// TIA Portal V19 export
FUNCTION "PREMIXING TRANSFER CYCLE" : Void   // FC25, LAD
{ S7_Optimized_Access := 'TRUE' }
// stored: SetENOAutomatically false
   VAR_TEMP   // added for the SCL form of the ladder/FBD networks
      _w1 : Bool;
   END_VAR
BEGIN

REGION Network 1: TRANSFER SELECT
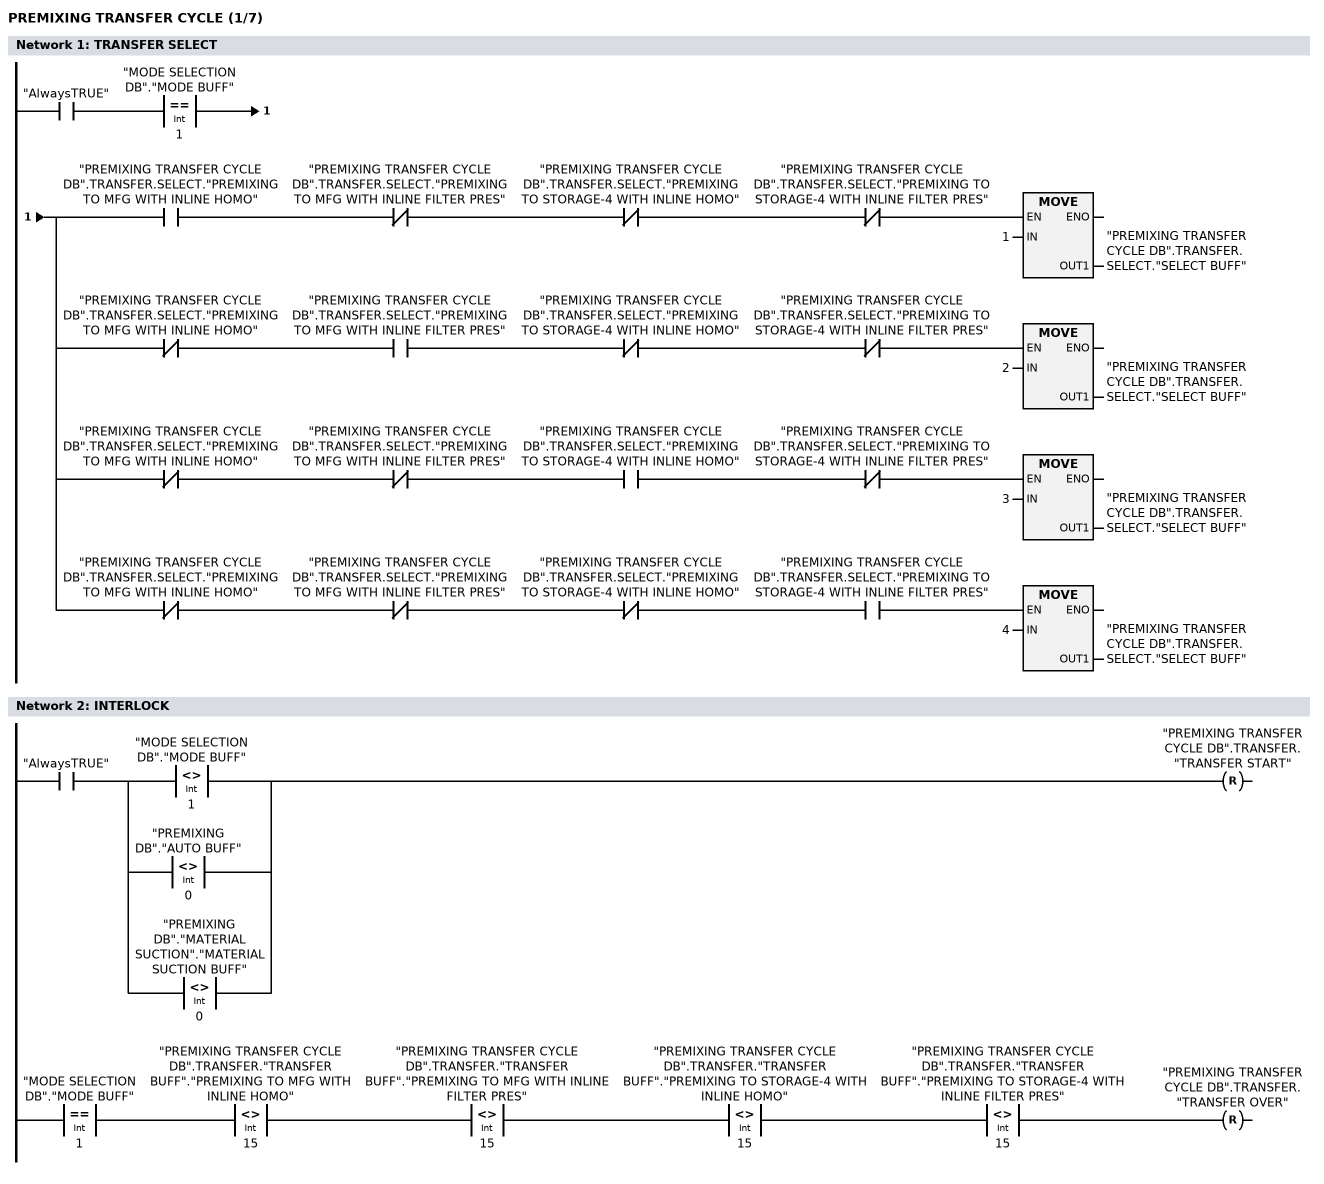
   RUNG wire#powerrail
      Contact( "AlwaysTRUE" )
      { S7_Templates := "SrcType := Int" } EQ_Contact(in1 := "MODE SELECTION DB"."MODE BUFF", in2 := 1)
      wire#w1
      Contact( "PREMIXING TRANSFER CYCLE DB".TRANSFER.SELECT."PREMIXING TO MFG WITH INLINE HOMO" )
      I_Contact( "PREMIXING TRANSFER CYCLE DB".TRANSFER.SELECT."PREMIXING TO MFG WITH INLINE FILTER PRES" )
      I_Contact( "PREMIXING TRANSFER CYCLE DB".TRANSFER.SELECT."PREMIXING TO STORAGE-4 WITH INLINE HOMO" )
      I_Contact( "PREMIXING TRANSFER CYCLE DB".TRANSFER.SELECT."PREMIXING TO STORAGE-4 WITH INLINE FILTER PRES" )
      Move(in := 1, out1 => "PREMIXING TRANSFER CYCLE DB".TRANSFER.SELECT."SELECT BUFF")
   END_RUNG
   RUNG wire#w1
      I_Contact( "PREMIXING TRANSFER CYCLE DB".TRANSFER.SELECT."PREMIXING TO MFG WITH INLINE HOMO" )
      Contact( "PREMIXING TRANSFER CYCLE DB".TRANSFER.SELECT."PREMIXING TO MFG WITH INLINE FILTER PRES" )
      I_Contact( "PREMIXING TRANSFER CYCLE DB".TRANSFER.SELECT."PREMIXING TO STORAGE-4 WITH INLINE HOMO" )
      I_Contact( "PREMIXING TRANSFER CYCLE DB".TRANSFER.SELECT."PREMIXING TO STORAGE-4 WITH INLINE FILTER PRES" )
      Move(in := 2, out1 => "PREMIXING TRANSFER CYCLE DB".TRANSFER.SELECT."SELECT BUFF")
   END_RUNG
   RUNG wire#w1
      I_Contact( "PREMIXING TRANSFER CYCLE DB".TRANSFER.SELECT."PREMIXING TO MFG WITH INLINE HOMO" )
      I_Contact( "PREMIXING TRANSFER CYCLE DB".TRANSFER.SELECT."PREMIXING TO MFG WITH INLINE FILTER PRES" )
      Contact( "PREMIXING TRANSFER CYCLE DB".TRANSFER.SELECT."PREMIXING TO STORAGE-4 WITH INLINE HOMO" )
      I_Contact( "PREMIXING TRANSFER CYCLE DB".TRANSFER.SELECT."PREMIXING TO STORAGE-4 WITH INLINE FILTER PRES" )
      Move(in := 3, out1 => "PREMIXING TRANSFER CYCLE DB".TRANSFER.SELECT."SELECT BUFF")
   END_RUNG
   RUNG wire#w1
      I_Contact( "PREMIXING TRANSFER CYCLE DB".TRANSFER.SELECT."PREMIXING TO MFG WITH INLINE HOMO" )
      I_Contact( "PREMIXING TRANSFER CYCLE DB".TRANSFER.SELECT."PREMIXING TO MFG WITH INLINE FILTER PRES" )
      I_Contact( "PREMIXING TRANSFER CYCLE DB".TRANSFER.SELECT."PREMIXING TO STORAGE-4 WITH INLINE HOMO" )
      Contact( "PREMIXING TRANSFER CYCLE DB".TRANSFER.SELECT."PREMIXING TO STORAGE-4 WITH INLINE FILTER PRES" )
      Move(in := 4, out1 => "PREMIXING TRANSFER CYCLE DB".TRANSFER.SELECT."SELECT BUFF")
   END_RUNG
   // the same network as SCL:
   #_w1 := "AlwaysTRUE" AND ("MODE SELECTION DB"."MODE BUFF" = 1);
   IF #_w1 AND "PREMIXING TRANSFER CYCLE DB".TRANSFER.SELECT."PREMIXING TO MFG WITH INLINE HOMO" AND NOT "PREMIXING TRANSFER CYCLE DB".TRANSFER.SELECT."PREMIXING TO MFG WITH INLINE FILTER PRES" AND NOT "PREMIXING TRANSFER CYCLE DB".TRANSFER.SELECT."PREMIXING TO STORAGE-4 WITH INLINE HOMO" AND NOT "PREMIXING TRANSFER CYCLE DB".TRANSFER.SELECT."PREMIXING TO STORAGE-4 WITH INLINE FILTER PRES" THEN
       "PREMIXING TRANSFER CYCLE DB".TRANSFER.SELECT."SELECT BUFF" := 1;
   END_IF;
   IF #_w1 AND NOT "PREMIXING TRANSFER CYCLE DB".TRANSFER.SELECT."PREMIXING TO MFG WITH INLINE HOMO" AND "PREMIXING TRANSFER CYCLE DB".TRANSFER.SELECT."PREMIXING TO MFG WITH INLINE FILTER PRES" AND NOT "PREMIXING TRANSFER CYCLE DB".TRANSFER.SELECT."PREMIXING TO STORAGE-4 WITH INLINE HOMO" AND NOT "PREMIXING TRANSFER CYCLE DB".TRANSFER.SELECT."PREMIXING TO STORAGE-4 WITH INLINE FILTER PRES" THEN
       "PREMIXING TRANSFER CYCLE DB".TRANSFER.SELECT."SELECT BUFF" := 2;
   END_IF;
   IF #_w1 AND NOT "PREMIXING TRANSFER CYCLE DB".TRANSFER.SELECT."PREMIXING TO MFG WITH INLINE HOMO" AND NOT "PREMIXING TRANSFER CYCLE DB".TRANSFER.SELECT."PREMIXING TO MFG WITH INLINE FILTER PRES" AND "PREMIXING TRANSFER CYCLE DB".TRANSFER.SELECT."PREMIXING TO STORAGE-4 WITH INLINE HOMO" AND NOT "PREMIXING TRANSFER CYCLE DB".TRANSFER.SELECT."PREMIXING TO STORAGE-4 WITH INLINE FILTER PRES" THEN
       "PREMIXING TRANSFER CYCLE DB".TRANSFER.SELECT."SELECT BUFF" := 3;
   END_IF;
   IF #_w1 AND NOT "PREMIXING TRANSFER CYCLE DB".TRANSFER.SELECT."PREMIXING TO MFG WITH INLINE HOMO" AND NOT "PREMIXING TRANSFER CYCLE DB".TRANSFER.SELECT."PREMIXING TO MFG WITH INLINE FILTER PRES" AND NOT "PREMIXING TRANSFER CYCLE DB".TRANSFER.SELECT."PREMIXING TO STORAGE-4 WITH INLINE HOMO" AND "PREMIXING TRANSFER CYCLE DB".TRANSFER.SELECT."PREMIXING TO STORAGE-4 WITH INLINE FILTER PRES" THEN
       "PREMIXING TRANSFER CYCLE DB".TRANSFER.SELECT."SELECT BUFF" := 4;
   END_IF;
END_REGION

REGION Network 2: INTERLOCK
   RUNG wire#powerrail
      Contact( "AlwaysTRUE" )
      wire#w1
      { S7_Templates := "SrcType := Int" } NE_Contact(in1 := "MODE SELECTION DB"."MODE BUFF", in2 := 1)
      wire#w2
      R_Coil( "PREMIXING TRANSFER CYCLE DB".TRANSFER."TRANSFER START" )
   END_RUNG
   RUNG wire#w1
      { S7_Templates := "SrcType := Int" } NE_Contact(in1 := "PREMIXING DB"."AUTO BUFF", in2 := 0)
   END_RUNG wire#w2
   RUNG wire#w1
      { S7_Templates := "SrcType := Int" } NE_Contact(in1 := "PREMIXING DB"."MATERIAL SUCTION"."MATERIAL SUCTION BUFF", in2 := 0)
   END_RUNG wire#w2
   RUNG wire#powerrail
      { S7_Templates := "SrcType := Int" } EQ_Contact(in1 := "MODE SELECTION DB"."MODE BUFF", in2 := 1)
      { S7_Templates := "SrcType := Int" } NE_Contact(in1 := "PREMIXING TRANSFER CYCLE DB".TRANSFER."TRANSFER BUFF"."PREMIXING TO MFG WITH INLINE HOMO", in2 := 15)
      { S7_Templates := "SrcType := Int" } NE_Contact(in1 := "PREMIXING TRANSFER CYCLE DB".TRANSFER."TRANSFER BUFF"."PREMIXING TO MFG WITH INLINE FILTER PRES", in2 := 15)
      { S7_Templates := "SrcType := Int" } NE_Contact(in1 := "PREMIXING TRANSFER CYCLE DB".TRANSFER."TRANSFER BUFF"."PREMIXING TO STORAGE-4 WITH INLINE HOMO", in2 := 15)
      { S7_Templates := "SrcType := Int" } NE_Contact(in1 := "PREMIXING TRANSFER CYCLE DB".TRANSFER."TRANSFER BUFF"."PREMIXING TO STORAGE-4 WITH INLINE FILTER PRES", in2 := 15)
      R_Coil( "PREMIXING TRANSFER CYCLE DB".TRANSFER."TRANSFER OVER" )
   END_RUNG
   // the same network as SCL:
   IF "AlwaysTRUE" AND (("MODE SELECTION DB"."MODE BUFF" <> 1) OR ("PREMIXING DB"."AUTO BUFF" <> 0) OR ("PREMIXING DB"."MATERIAL SUCTION"."MATERIAL SUCTION BUFF" <> 0)) THEN
       "PREMIXING TRANSFER CYCLE DB".TRANSFER."TRANSFER START" := FALSE;
   END_IF;
   IF ("MODE SELECTION DB"."MODE BUFF" = 1) AND ("PREMIXING TRANSFER CYCLE DB".TRANSFER."TRANSFER BUFF"."PREMIXING TO MFG WITH INLINE HOMO" <> 15) AND ("PREMIXING TRANSFER CYCLE DB".TRANSFER."TRANSFER BUFF"."PREMIXING TO MFG WITH INLINE FILTER PRES" <> 15) AND ("PREMIXING TRANSFER CYCLE DB".TRANSFER."TRANSFER BUFF"."PREMIXING TO STORAGE-4 WITH INLINE HOMO" <> 15) AND ("PREMIXING TRANSFER CYCLE DB".TRANSFER."TRANSFER BUFF"."PREMIXING TO STORAGE-4 WITH INLINE FILTER PRES" <> 15) THEN
       "PREMIXING TRANSFER CYCLE DB".TRANSFER."TRANSFER OVER" := FALSE;
   END_IF;
END_REGION

REGION Network 3: TRANSFER START ///////////////////////////// PREMIXING TO MFG WITH INLINE HOMO
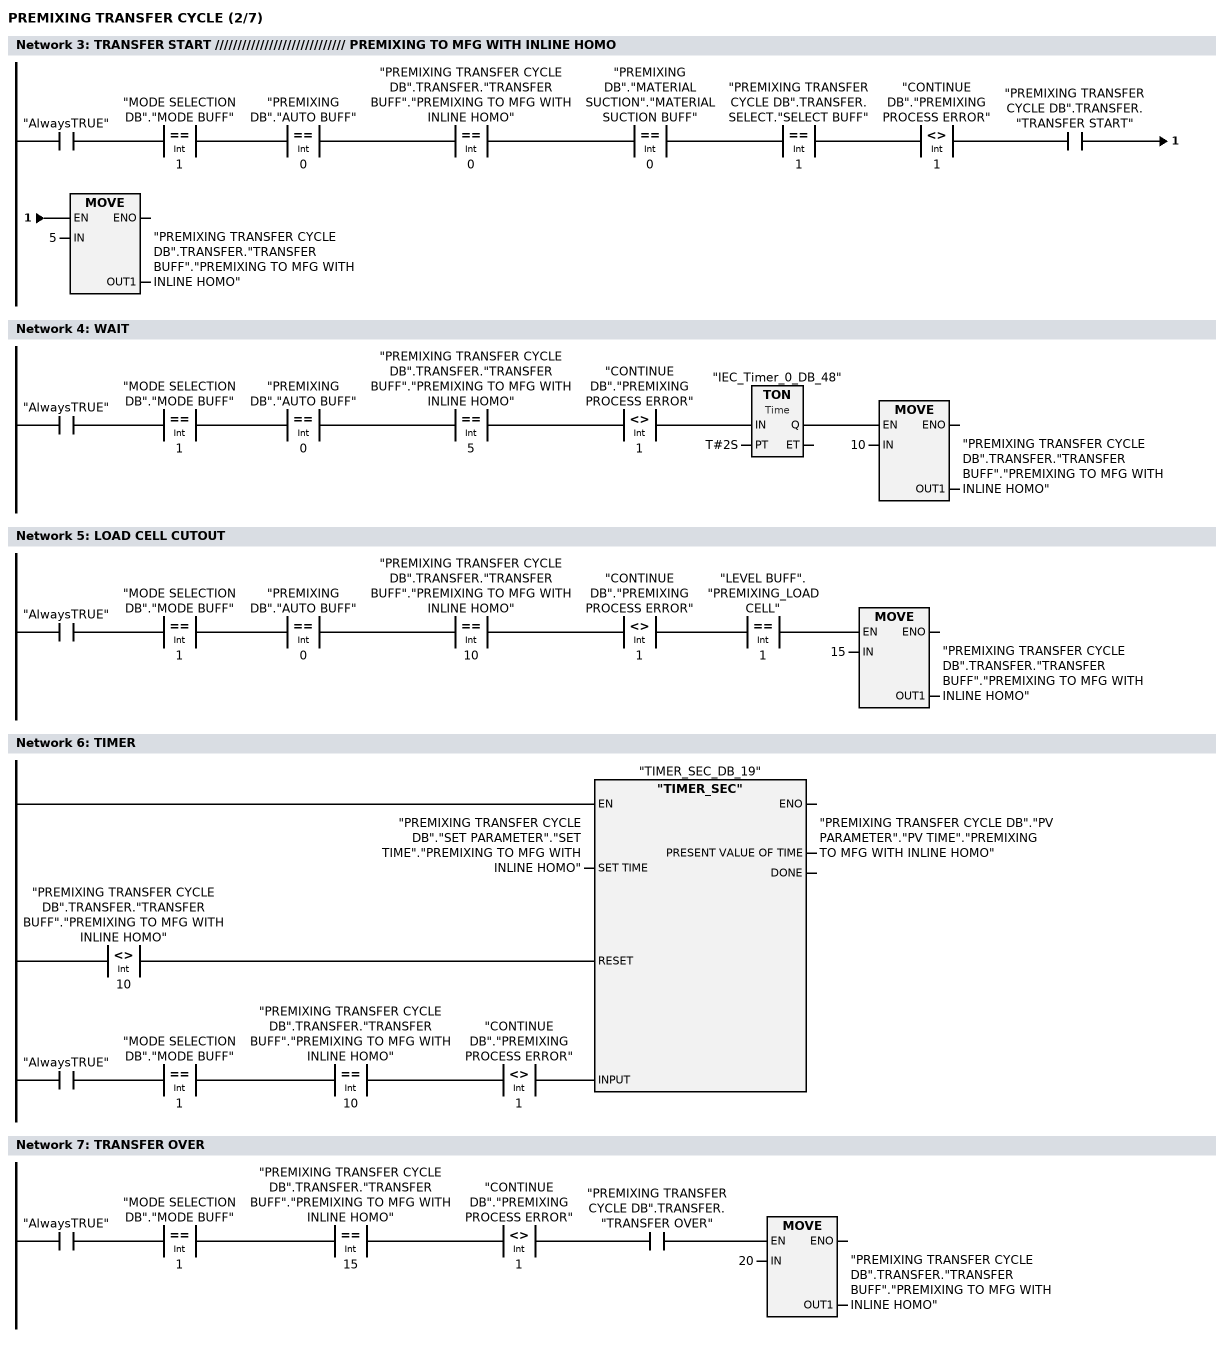
   RUNG wire#powerrail
      Contact( "AlwaysTRUE" )
      { S7_Templates := "SrcType := Int" } EQ_Contact(in1 := "MODE SELECTION DB"."MODE BUFF", in2 := 1)
      { S7_Templates := "SrcType := Int" } EQ_Contact(in1 := "PREMIXING DB"."AUTO BUFF", in2 := 0)
      { S7_Templates := "SrcType := Int" } EQ_Contact(in1 := "PREMIXING TRANSFER CYCLE DB".TRANSFER."TRANSFER BUFF"."PREMIXING TO MFG WITH INLINE HOMO", in2 := 0)
      { S7_Templates := "SrcType := Int" } EQ_Contact(in1 := "PREMIXING DB"."MATERIAL SUCTION"."MATERIAL SUCTION BUFF", in2 := 0)
      { S7_Templates := "SrcType := Int" } EQ_Contact(in1 := "PREMIXING TRANSFER CYCLE DB".TRANSFER.SELECT."SELECT BUFF", in2 := 1)
      { S7_Templates := "SrcType := Int" } NE_Contact(in1 := "CONTINUE DB"."PREMIXING PROCESS ERROR", in2 := 1)
      Contact( "PREMIXING TRANSFER CYCLE DB".TRANSFER."TRANSFER START" )
      Move(in := 5, out1 => "PREMIXING TRANSFER CYCLE DB".TRANSFER."TRANSFER BUFF"."PREMIXING TO MFG WITH INLINE HOMO")
   END_RUNG
   // the same network as SCL:
   IF "AlwaysTRUE" AND ("MODE SELECTION DB"."MODE BUFF" = 1) AND ("PREMIXING DB"."AUTO BUFF" = 0) AND ("PREMIXING TRANSFER CYCLE DB".TRANSFER."TRANSFER BUFF"."PREMIXING TO MFG WITH INLINE HOMO" = 0) AND ("PREMIXING DB"."MATERIAL SUCTION"."MATERIAL SUCTION BUFF" = 0) AND ("PREMIXING TRANSFER CYCLE DB".TRANSFER.SELECT."SELECT BUFF" = 1) AND ("CONTINUE DB"."PREMIXING PROCESS ERROR" <> 1) AND "PREMIXING TRANSFER CYCLE DB".TRANSFER."TRANSFER START" THEN
       "PREMIXING TRANSFER CYCLE DB".TRANSFER."TRANSFER BUFF"."PREMIXING TO MFG WITH INLINE HOMO" := 5;
   END_IF;
END_REGION

REGION Network 4: WAIT
   RUNG wire#powerrail
      Contact( "AlwaysTRUE" )
      { S7_Templates := "SrcType := Int" } EQ_Contact(in1 := "MODE SELECTION DB"."MODE BUFF", in2 := 1)
      { S7_Templates := "SrcType := Int" } EQ_Contact(in1 := "PREMIXING DB"."AUTO BUFF", in2 := 0)
      { S7_Templates := "SrcType := Int" } EQ_Contact(in1 := "PREMIXING TRANSFER CYCLE DB".TRANSFER."TRANSFER BUFF"."PREMIXING TO MFG WITH INLINE HOMO", in2 := 5)
      { S7_Templates := "SrcType := Int" } NE_Contact(in1 := "CONTINUE DB"."PREMIXING PROCESS ERROR", in2 := 1)
      { S7_Templates := "time_type := Time" } "IEC_Timer_0_DB_48".TON(pt := T#2S, et =>)
      Move(in := 10, out1 => "PREMIXING TRANSFER CYCLE DB".TRANSFER."TRANSFER BUFF"."PREMIXING TO MFG WITH INLINE HOMO")
   END_RUNG
   // the same network as SCL:
   "IEC_Timer_0_DB_48".TON(IN := "AlwaysTRUE" AND ("MODE SELECTION DB"."MODE BUFF" = 1) AND ("PREMIXING DB"."AUTO BUFF" = 0) AND ("PREMIXING TRANSFER CYCLE DB".TRANSFER."TRANSFER BUFF"."PREMIXING TO MFG WITH INLINE HOMO" = 5) AND ("CONTINUE DB"."PREMIXING PROCESS ERROR" <> 1),
                           PT := T#2S);
   IF "IEC_Timer_0_DB_48".Q THEN
       "PREMIXING TRANSFER CYCLE DB".TRANSFER."TRANSFER BUFF"."PREMIXING TO MFG WITH INLINE HOMO" := 10;
   END_IF;
END_REGION

REGION Network 5: LOAD CELL CUTOUT
   RUNG wire#powerrail
      Contact( "AlwaysTRUE" )
      { S7_Templates := "SrcType := Int" } EQ_Contact(in1 := "MODE SELECTION DB"."MODE BUFF", in2 := 1)
      { S7_Templates := "SrcType := Int" } EQ_Contact(in1 := "PREMIXING DB"."AUTO BUFF", in2 := 0)
      { S7_Templates := "SrcType := Int" } EQ_Contact(in1 := "PREMIXING TRANSFER CYCLE DB".TRANSFER."TRANSFER BUFF"."PREMIXING TO MFG WITH INLINE HOMO", in2 := 10)
      { S7_Templates := "SrcType := Int" } NE_Contact(in1 := "CONTINUE DB"."PREMIXING PROCESS ERROR", in2 := 1)
      { S7_Templates := "SrcType := Int" } EQ_Contact(in1 := "LEVEL BUFF"."PREMIXING_LOAD CELL", in2 := 1)
      Move(in := 15, out1 => "PREMIXING TRANSFER CYCLE DB".TRANSFER."TRANSFER BUFF"."PREMIXING TO MFG WITH INLINE HOMO")
   END_RUNG
   // the same network as SCL:
   IF "AlwaysTRUE" AND ("MODE SELECTION DB"."MODE BUFF" = 1) AND ("PREMIXING DB"."AUTO BUFF" = 0) AND ("PREMIXING TRANSFER CYCLE DB".TRANSFER."TRANSFER BUFF"."PREMIXING TO MFG WITH INLINE HOMO" = 10) AND ("CONTINUE DB"."PREMIXING PROCESS ERROR" <> 1) AND ("LEVEL BUFF"."PREMIXING_LOAD CELL" = 1) THEN
       "PREMIXING TRANSFER CYCLE DB".TRANSFER."TRANSFER BUFF"."PREMIXING TO MFG WITH INLINE HOMO" := 15;
   END_IF;
END_REGION

REGION Network 6: TIMER
   RUNG wire#powerrail
      "TIMER_SEC_DB_19"(RESET := wire#w1, INPUT := wire#w2, "SET TIME" := "PREMIXING TRANSFER CYCLE DB"."SET PARAMETER"."SET TIME"."PREMIXING TO MFG WITH INLINE HOMO", "PRESENT VALUE OF TIME" => "PREMIXING TRANSFER CYCLE DB"."PV PARAMETER"."PV TIME"."PREMIXING TO MFG WITH INLINE HOMO", DONE =>)
   END_RUNG
   RUNG wire#powerrail
      { S7_Templates := "SrcType := Int" } NE_Contact(in1 := "PREMIXING TRANSFER CYCLE DB".TRANSFER."TRANSFER BUFF"."PREMIXING TO MFG WITH INLINE HOMO", in2 := 10)
   END_RUNG wire#w1
   RUNG wire#powerrail
      Contact( "AlwaysTRUE" )
      { S7_Templates := "SrcType := Int" } EQ_Contact(in1 := "MODE SELECTION DB"."MODE BUFF", in2 := 1)
      { S7_Templates := "SrcType := Int" } EQ_Contact(in1 := "PREMIXING TRANSFER CYCLE DB".TRANSFER."TRANSFER BUFF"."PREMIXING TO MFG WITH INLINE HOMO", in2 := 10)
      { S7_Templates := "SrcType := Int" } NE_Contact(in1 := "CONTINUE DB"."PREMIXING PROCESS ERROR", in2 := 1)
   END_RUNG wire#w2
   // the same network as SCL:
   "TIMER_SEC_DB_19"("SET TIME" := "PREMIXING TRANSFER CYCLE DB"."SET PARAMETER"."SET TIME"."PREMIXING TO MFG WITH INLINE HOMO",   // "TIMER_SEC"
                     RESET := "PREMIXING TRANSFER CYCLE DB".TRANSFER."TRANSFER BUFF"."PREMIXING TO MFG WITH INLINE HOMO" <> 10,
                     INPUT := "AlwaysTRUE" AND ("MODE SELECTION DB"."MODE BUFF" = 1) AND ("PREMIXING TRANSFER CYCLE DB".TRANSFER."TRANSFER BUFF"."PREMIXING TO MFG WITH INLINE HOMO" = 10) AND ("CONTINUE DB"."PREMIXING PROCESS ERROR" <> 1),
                     "PRESENT VALUE OF TIME" => "PREMIXING TRANSFER CYCLE DB"."PV PARAMETER"."PV TIME"."PREMIXING TO MFG WITH INLINE HOMO");
END_REGION

REGION Network 7: TRANSFER OVER
   RUNG wire#powerrail
      Contact( "AlwaysTRUE" )
      { S7_Templates := "SrcType := Int" } EQ_Contact(in1 := "MODE SELECTION DB"."MODE BUFF", in2 := 1)
      { S7_Templates := "SrcType := Int" } EQ_Contact(in1 := "PREMIXING TRANSFER CYCLE DB".TRANSFER."TRANSFER BUFF"."PREMIXING TO MFG WITH INLINE HOMO", in2 := 15)
      { S7_Templates := "SrcType := Int" } NE_Contact(in1 := "CONTINUE DB"."PREMIXING PROCESS ERROR", in2 := 1)
      Contact( "PREMIXING TRANSFER CYCLE DB".TRANSFER."TRANSFER OVER" )
      Move(in := 20, out1 => "PREMIXING TRANSFER CYCLE DB".TRANSFER."TRANSFER BUFF"."PREMIXING TO MFG WITH INLINE HOMO")
   END_RUNG
   // the same network as SCL:
   IF "AlwaysTRUE" AND ("MODE SELECTION DB"."MODE BUFF" = 1) AND ("PREMIXING TRANSFER CYCLE DB".TRANSFER."TRANSFER BUFF"."PREMIXING TO MFG WITH INLINE HOMO" = 15) AND ("CONTINUE DB"."PREMIXING PROCESS ERROR" <> 1) AND "PREMIXING TRANSFER CYCLE DB".TRANSFER."TRANSFER OVER" THEN
       "PREMIXING TRANSFER CYCLE DB".TRANSFER."TRANSFER BUFF"."PREMIXING TO MFG WITH INLINE HOMO" := 20;
   END_IF;
END_REGION

REGION Network 8: STOP
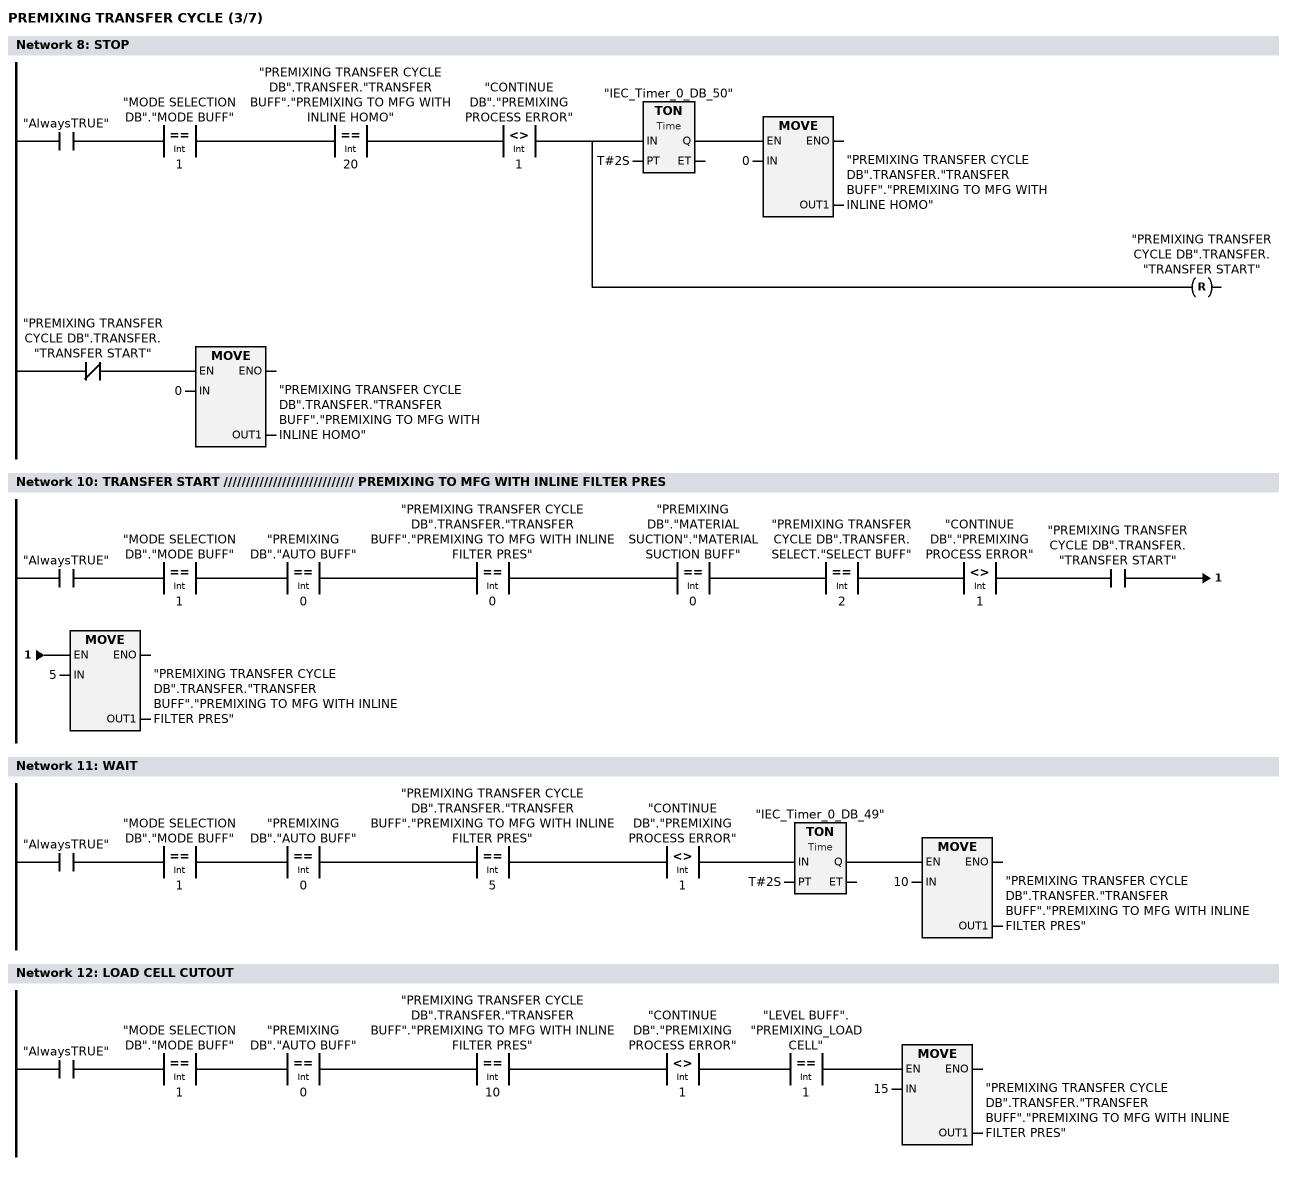
   RUNG wire#powerrail
      Contact( "AlwaysTRUE" )
      { S7_Templates := "SrcType := Int" } EQ_Contact(in1 := "MODE SELECTION DB"."MODE BUFF", in2 := 1)
      { S7_Templates := "SrcType := Int" } EQ_Contact(in1 := "PREMIXING TRANSFER CYCLE DB".TRANSFER."TRANSFER BUFF"."PREMIXING TO MFG WITH INLINE HOMO", in2 := 20)
      { S7_Templates := "SrcType := Int" } NE_Contact(in1 := "CONTINUE DB"."PREMIXING PROCESS ERROR", in2 := 1)
      wire#w1
      { S7_Templates := "time_type := Time" } "IEC_Timer_0_DB_50".TON(pt := T#2S, et =>)
      Move(in := 0, out1 => "PREMIXING TRANSFER CYCLE DB".TRANSFER."TRANSFER BUFF"."PREMIXING TO MFG WITH INLINE HOMO")
   END_RUNG
   RUNG wire#w1
      R_Coil( "PREMIXING TRANSFER CYCLE DB".TRANSFER."TRANSFER START" )
   END_RUNG
   RUNG wire#powerrail
      I_Contact( "PREMIXING TRANSFER CYCLE DB".TRANSFER."TRANSFER START" )
      Move(in := 0, out1 => "PREMIXING TRANSFER CYCLE DB".TRANSFER."TRANSFER BUFF"."PREMIXING TO MFG WITH INLINE HOMO")
   END_RUNG
   // the same network as SCL:
   #_w1 := "AlwaysTRUE" AND ("MODE SELECTION DB"."MODE BUFF" = 1) AND ("PREMIXING TRANSFER CYCLE DB".TRANSFER."TRANSFER BUFF"."PREMIXING TO MFG WITH INLINE HOMO" = 20) AND ("CONTINUE DB"."PREMIXING PROCESS ERROR" <> 1);
   "IEC_Timer_0_DB_50".TON(IN := #_w1, PT := T#2S);
   IF "IEC_Timer_0_DB_50".Q THEN
       "PREMIXING TRANSFER CYCLE DB".TRANSFER."TRANSFER BUFF"."PREMIXING TO MFG WITH INLINE HOMO" := 0;
   END_IF;
   IF #_w1 THEN "PREMIXING TRANSFER CYCLE DB".TRANSFER."TRANSFER START" := FALSE; END_IF;
   IF NOT "PREMIXING TRANSFER CYCLE DB".TRANSFER."TRANSFER START" THEN
       "PREMIXING TRANSFER CYCLE DB".TRANSFER."TRANSFER BUFF"."PREMIXING TO MFG WITH INLINE HOMO" := 0;
   END_IF;
END_REGION

REGION Network 10: TRANSFER START ///////////////////////////// PREMIXING TO MFG WITH INLINE FILTER PRES
   RUNG wire#powerrail
      Contact( "AlwaysTRUE" )
      { S7_Templates := "SrcType := Int" } EQ_Contact(in1 := "MODE SELECTION DB"."MODE BUFF", in2 := 1)
      { S7_Templates := "SrcType := Int" } EQ_Contact(in1 := "PREMIXING DB"."AUTO BUFF", in2 := 0)
      { S7_Templates := "SrcType := Int" } EQ_Contact(in1 := "PREMIXING TRANSFER CYCLE DB".TRANSFER."TRANSFER BUFF"."PREMIXING TO MFG WITH INLINE FILTER PRES", in2 := 0)
      { S7_Templates := "SrcType := Int" } EQ_Contact(in1 := "PREMIXING DB"."MATERIAL SUCTION"."MATERIAL SUCTION BUFF", in2 := 0)
      { S7_Templates := "SrcType := Int" } EQ_Contact(in1 := "PREMIXING TRANSFER CYCLE DB".TRANSFER.SELECT."SELECT BUFF", in2 := 2)
      { S7_Templates := "SrcType := Int" } NE_Contact(in1 := "CONTINUE DB"."PREMIXING PROCESS ERROR", in2 := 1)
      Contact( "PREMIXING TRANSFER CYCLE DB".TRANSFER."TRANSFER START" )
      Move(in := 5, out1 => "PREMIXING TRANSFER CYCLE DB".TRANSFER."TRANSFER BUFF"."PREMIXING TO MFG WITH INLINE FILTER PRES")
   END_RUNG
   // the same network as SCL:
   IF "AlwaysTRUE" AND ("MODE SELECTION DB"."MODE BUFF" = 1) AND ("PREMIXING DB"."AUTO BUFF" = 0) AND ("PREMIXING TRANSFER CYCLE DB".TRANSFER."TRANSFER BUFF"."PREMIXING TO MFG WITH INLINE FILTER PRES" = 0) AND ("PREMIXING DB"."MATERIAL SUCTION"."MATERIAL SUCTION BUFF" = 0) AND ("PREMIXING TRANSFER CYCLE DB".TRANSFER.SELECT."SELECT BUFF" = 2) AND ("CONTINUE DB"."PREMIXING PROCESS ERROR" <> 1) AND "PREMIXING TRANSFER CYCLE DB".TRANSFER."TRANSFER START" THEN
       "PREMIXING TRANSFER CYCLE DB".TRANSFER."TRANSFER BUFF"."PREMIXING TO MFG WITH INLINE FILTER PRES" := 5;
   END_IF;
END_REGION

REGION Network 11: WAIT
   RUNG wire#powerrail
      Contact( "AlwaysTRUE" )
      { S7_Templates := "SrcType := Int" } EQ_Contact(in1 := "MODE SELECTION DB"."MODE BUFF", in2 := 1)
      { S7_Templates := "SrcType := Int" } EQ_Contact(in1 := "PREMIXING DB"."AUTO BUFF", in2 := 0)
      { S7_Templates := "SrcType := Int" } EQ_Contact(in1 := "PREMIXING TRANSFER CYCLE DB".TRANSFER."TRANSFER BUFF"."PREMIXING TO MFG WITH INLINE FILTER PRES", in2 := 5)
      { S7_Templates := "SrcType := Int" } NE_Contact(in1 := "CONTINUE DB"."PREMIXING PROCESS ERROR", in2 := 1)
      { S7_Templates := "time_type := Time" } "IEC_Timer_0_DB_49".TON(pt := T#2S, et =>)
      Move(in := 10, out1 => "PREMIXING TRANSFER CYCLE DB".TRANSFER."TRANSFER BUFF"."PREMIXING TO MFG WITH INLINE FILTER PRES")
   END_RUNG
   // the same network as SCL:
   "IEC_Timer_0_DB_49".TON(IN := "AlwaysTRUE" AND ("MODE SELECTION DB"."MODE BUFF" = 1) AND ("PREMIXING DB"."AUTO BUFF" = 0) AND ("PREMIXING TRANSFER CYCLE DB".TRANSFER."TRANSFER BUFF"."PREMIXING TO MFG WITH INLINE FILTER PRES" = 5) AND ("CONTINUE DB"."PREMIXING PROCESS ERROR" <> 1),
                           PT := T#2S);
   IF "IEC_Timer_0_DB_49".Q THEN
       "PREMIXING TRANSFER CYCLE DB".TRANSFER."TRANSFER BUFF"."PREMIXING TO MFG WITH INLINE FILTER PRES" := 10;
   END_IF;
END_REGION

REGION Network 12: LOAD CELL CUTOUT
   RUNG wire#powerrail
      Contact( "AlwaysTRUE" )
      { S7_Templates := "SrcType := Int" } EQ_Contact(in1 := "MODE SELECTION DB"."MODE BUFF", in2 := 1)
      { S7_Templates := "SrcType := Int" } EQ_Contact(in1 := "PREMIXING DB"."AUTO BUFF", in2 := 0)
      { S7_Templates := "SrcType := Int" } EQ_Contact(in1 := "PREMIXING TRANSFER CYCLE DB".TRANSFER."TRANSFER BUFF"."PREMIXING TO MFG WITH INLINE FILTER PRES", in2 := 10)
      { S7_Templates := "SrcType := Int" } NE_Contact(in1 := "CONTINUE DB"."PREMIXING PROCESS ERROR", in2 := 1)
      { S7_Templates := "SrcType := Int" } EQ_Contact(in1 := "LEVEL BUFF"."PREMIXING_LOAD CELL", in2 := 1)
      Move(in := 15, out1 => "PREMIXING TRANSFER CYCLE DB".TRANSFER."TRANSFER BUFF"."PREMIXING TO MFG WITH INLINE FILTER PRES")
   END_RUNG
   // the same network as SCL:
   IF "AlwaysTRUE" AND ("MODE SELECTION DB"."MODE BUFF" = 1) AND ("PREMIXING DB"."AUTO BUFF" = 0) AND ("PREMIXING TRANSFER CYCLE DB".TRANSFER."TRANSFER BUFF"."PREMIXING TO MFG WITH INLINE FILTER PRES" = 10) AND ("CONTINUE DB"."PREMIXING PROCESS ERROR" <> 1) AND ("LEVEL BUFF"."PREMIXING_LOAD CELL" = 1) THEN
       "PREMIXING TRANSFER CYCLE DB".TRANSFER."TRANSFER BUFF"."PREMIXING TO MFG WITH INLINE FILTER PRES" := 15;
   END_IF;
END_REGION

REGION Network 13: TIMER
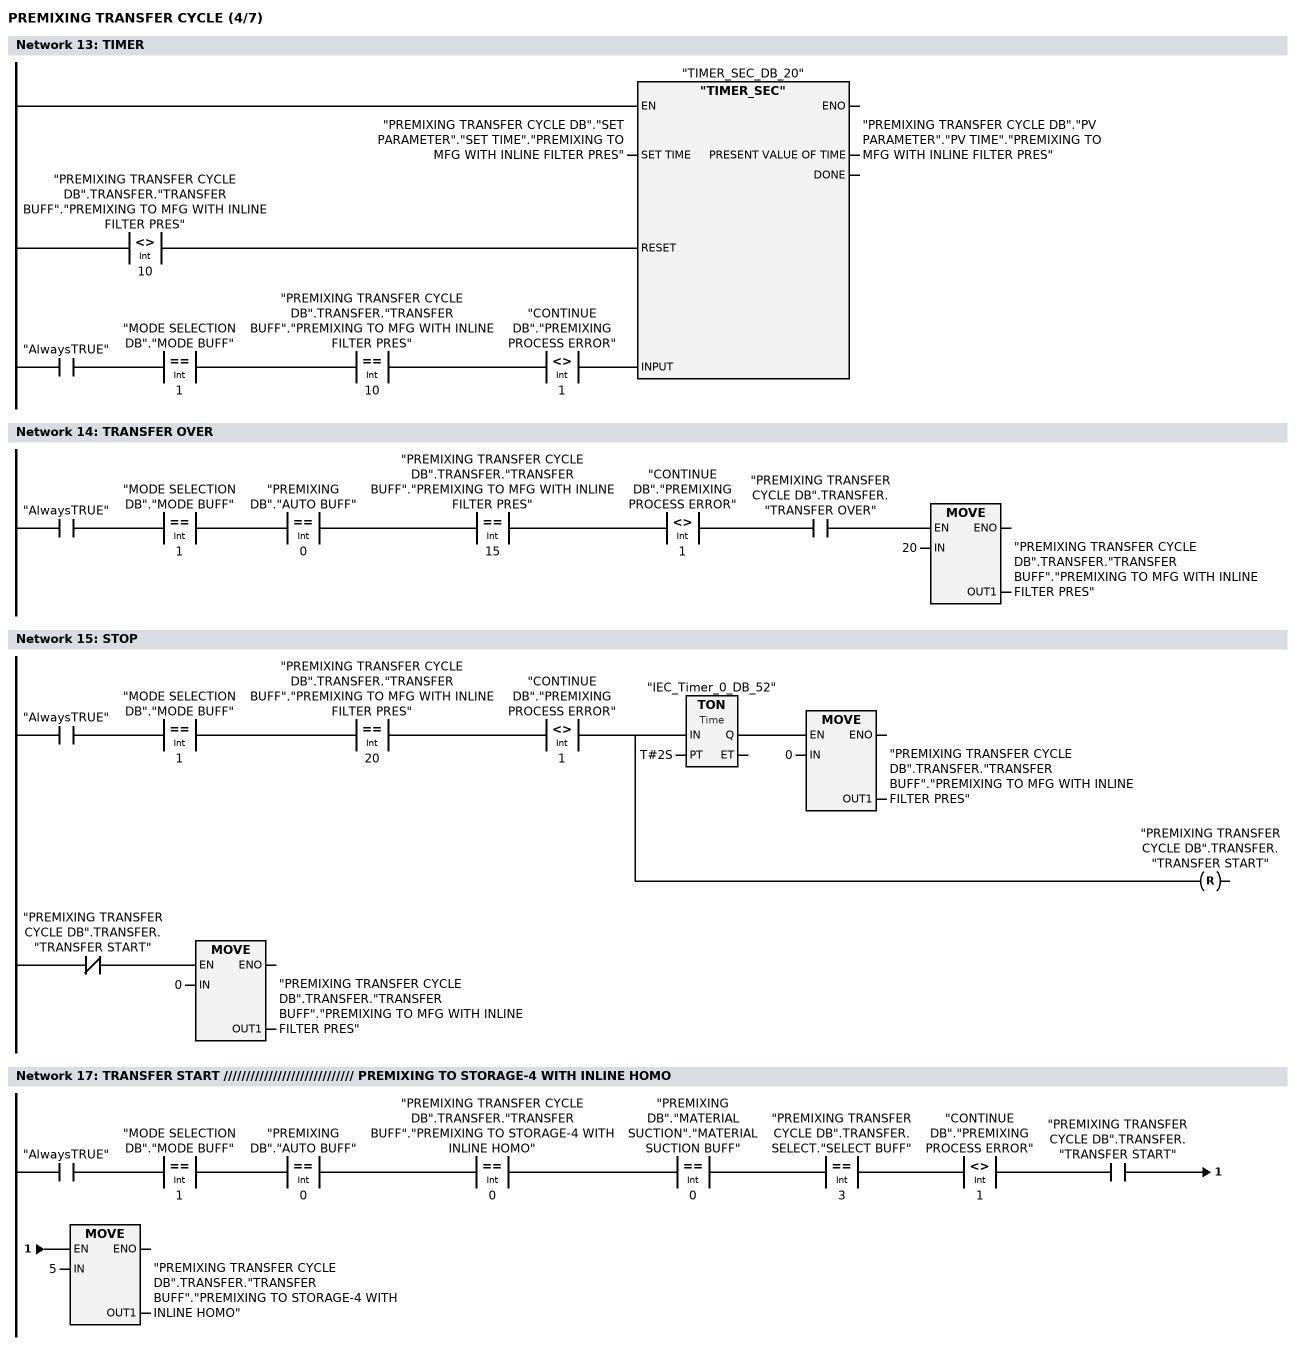
   RUNG wire#powerrail
      "TIMER_SEC_DB_20"(RESET := wire#w1, INPUT := wire#w2, "SET TIME" := "PREMIXING TRANSFER CYCLE DB"."SET PARAMETER"."SET TIME"."PREMIXING TO MFG WITH INLINE FILTER PRES", "PRESENT VALUE OF TIME" => "PREMIXING TRANSFER CYCLE DB"."PV PARAMETER"."PV TIME"."PREMIXING TO MFG WITH INLINE FILTER PRES", DONE =>)
   END_RUNG
   RUNG wire#powerrail
      { S7_Templates := "SrcType := Int" } NE_Contact(in1 := "PREMIXING TRANSFER CYCLE DB".TRANSFER."TRANSFER BUFF"."PREMIXING TO MFG WITH INLINE FILTER PRES", in2 := 10)
   END_RUNG wire#w1
   RUNG wire#powerrail
      Contact( "AlwaysTRUE" )
      { S7_Templates := "SrcType := Int" } EQ_Contact(in1 := "MODE SELECTION DB"."MODE BUFF", in2 := 1)
      { S7_Templates := "SrcType := Int" } EQ_Contact(in1 := "PREMIXING TRANSFER CYCLE DB".TRANSFER."TRANSFER BUFF"."PREMIXING TO MFG WITH INLINE FILTER PRES", in2 := 10)
      { S7_Templates := "SrcType := Int" } NE_Contact(in1 := "CONTINUE DB"."PREMIXING PROCESS ERROR", in2 := 1)
   END_RUNG wire#w2
   // the same network as SCL:
   "TIMER_SEC_DB_20"("SET TIME" := "PREMIXING TRANSFER CYCLE DB"."SET PARAMETER"."SET TIME"."PREMIXING TO MFG WITH INLINE FILTER PRES",   // "TIMER_SEC"
                     RESET := "PREMIXING TRANSFER CYCLE DB".TRANSFER."TRANSFER BUFF"."PREMIXING TO MFG WITH INLINE FILTER PRES" <> 10,
                     INPUT := "AlwaysTRUE" AND ("MODE SELECTION DB"."MODE BUFF" = 1) AND ("PREMIXING TRANSFER CYCLE DB".TRANSFER."TRANSFER BUFF"."PREMIXING TO MFG WITH INLINE FILTER PRES" = 10) AND ("CONTINUE DB"."PREMIXING PROCESS ERROR" <> 1),
                     "PRESENT VALUE OF TIME" => "PREMIXING TRANSFER CYCLE DB"."PV PARAMETER"."PV TIME"."PREMIXING TO MFG WITH INLINE FILTER PRES");
END_REGION

REGION Network 14: TRANSFER OVER
   RUNG wire#powerrail
      Contact( "AlwaysTRUE" )
      { S7_Templates := "SrcType := Int" } EQ_Contact(in1 := "MODE SELECTION DB"."MODE BUFF", in2 := 1)
      { S7_Templates := "SrcType := Int" } EQ_Contact(in1 := "PREMIXING DB"."AUTO BUFF", in2 := 0)
      { S7_Templates := "SrcType := Int" } EQ_Contact(in1 := "PREMIXING TRANSFER CYCLE DB".TRANSFER."TRANSFER BUFF"."PREMIXING TO MFG WITH INLINE FILTER PRES", in2 := 15)
      { S7_Templates := "SrcType := Int" } NE_Contact(in1 := "CONTINUE DB"."PREMIXING PROCESS ERROR", in2 := 1)
      Contact( "PREMIXING TRANSFER CYCLE DB".TRANSFER."TRANSFER OVER" )
      Move(in := 20, out1 => "PREMIXING TRANSFER CYCLE DB".TRANSFER."TRANSFER BUFF"."PREMIXING TO MFG WITH INLINE FILTER PRES")
   END_RUNG
   // the same network as SCL:
   IF "AlwaysTRUE" AND ("MODE SELECTION DB"."MODE BUFF" = 1) AND ("PREMIXING DB"."AUTO BUFF" = 0) AND ("PREMIXING TRANSFER CYCLE DB".TRANSFER."TRANSFER BUFF"."PREMIXING TO MFG WITH INLINE FILTER PRES" = 15) AND ("CONTINUE DB"."PREMIXING PROCESS ERROR" <> 1) AND "PREMIXING TRANSFER CYCLE DB".TRANSFER."TRANSFER OVER" THEN
       "PREMIXING TRANSFER CYCLE DB".TRANSFER."TRANSFER BUFF"."PREMIXING TO MFG WITH INLINE FILTER PRES" := 20;
   END_IF;
END_REGION

REGION Network 15: STOP
   RUNG wire#powerrail
      Contact( "AlwaysTRUE" )
      { S7_Templates := "SrcType := Int" } EQ_Contact(in1 := "MODE SELECTION DB"."MODE BUFF", in2 := 1)
      { S7_Templates := "SrcType := Int" } EQ_Contact(in1 := "PREMIXING TRANSFER CYCLE DB".TRANSFER."TRANSFER BUFF"."PREMIXING TO MFG WITH INLINE FILTER PRES", in2 := 20)
      { S7_Templates := "SrcType := Int" } NE_Contact(in1 := "CONTINUE DB"."PREMIXING PROCESS ERROR", in2 := 1)
      wire#w1
      { S7_Templates := "time_type := Time" } "IEC_Timer_0_DB_52".TON(pt := T#2S, et =>)
      Move(in := 0, out1 => "PREMIXING TRANSFER CYCLE DB".TRANSFER."TRANSFER BUFF"."PREMIXING TO MFG WITH INLINE FILTER PRES")
   END_RUNG
   RUNG wire#w1
      R_Coil( "PREMIXING TRANSFER CYCLE DB".TRANSFER."TRANSFER START" )
   END_RUNG
   RUNG wire#powerrail
      I_Contact( "PREMIXING TRANSFER CYCLE DB".TRANSFER."TRANSFER START" )
      Move(in := 0, out1 => "PREMIXING TRANSFER CYCLE DB".TRANSFER."TRANSFER BUFF"."PREMIXING TO MFG WITH INLINE FILTER PRES")
   END_RUNG
   // the same network as SCL:
   #_w1 := "AlwaysTRUE" AND ("MODE SELECTION DB"."MODE BUFF" = 1) AND ("PREMIXING TRANSFER CYCLE DB".TRANSFER."TRANSFER BUFF"."PREMIXING TO MFG WITH INLINE FILTER PRES" = 20) AND ("CONTINUE DB"."PREMIXING PROCESS ERROR" <> 1);
   "IEC_Timer_0_DB_52".TON(IN := #_w1, PT := T#2S);
   IF "IEC_Timer_0_DB_52".Q THEN
       "PREMIXING TRANSFER CYCLE DB".TRANSFER."TRANSFER BUFF"."PREMIXING TO MFG WITH INLINE FILTER PRES" := 0;
   END_IF;
   IF #_w1 THEN "PREMIXING TRANSFER CYCLE DB".TRANSFER."TRANSFER START" := FALSE; END_IF;
   IF NOT "PREMIXING TRANSFER CYCLE DB".TRANSFER."TRANSFER START" THEN
       "PREMIXING TRANSFER CYCLE DB".TRANSFER."TRANSFER BUFF"."PREMIXING TO MFG WITH INLINE FILTER PRES" := 0;
   END_IF;
END_REGION

REGION Network 17: TRANSFER START ///////////////////////////// PREMIXING TO STORAGE-4 WITH INLINE HOMO
   RUNG wire#powerrail
      Contact( "AlwaysTRUE" )
      { S7_Templates := "SrcType := Int" } EQ_Contact(in1 := "MODE SELECTION DB"."MODE BUFF", in2 := 1)
      { S7_Templates := "SrcType := Int" } EQ_Contact(in1 := "PREMIXING DB"."AUTO BUFF", in2 := 0)
      { S7_Templates := "SrcType := Int" } EQ_Contact(in1 := "PREMIXING TRANSFER CYCLE DB".TRANSFER."TRANSFER BUFF"."PREMIXING TO STORAGE-4 WITH INLINE HOMO", in2 := 0)
      { S7_Templates := "SrcType := Int" } EQ_Contact(in1 := "PREMIXING DB"."MATERIAL SUCTION"."MATERIAL SUCTION BUFF", in2 := 0)
      { S7_Templates := "SrcType := Int" } EQ_Contact(in1 := "PREMIXING TRANSFER CYCLE DB".TRANSFER.SELECT."SELECT BUFF", in2 := 3)
      { S7_Templates := "SrcType := Int" } NE_Contact(in1 := "CONTINUE DB"."PREMIXING PROCESS ERROR", in2 := 1)
      Contact( "PREMIXING TRANSFER CYCLE DB".TRANSFER."TRANSFER START" )
      Move(in := 5, out1 => "PREMIXING TRANSFER CYCLE DB".TRANSFER."TRANSFER BUFF"."PREMIXING TO STORAGE-4 WITH INLINE HOMO")
   END_RUNG
   // the same network as SCL:
   IF "AlwaysTRUE" AND ("MODE SELECTION DB"."MODE BUFF" = 1) AND ("PREMIXING DB"."AUTO BUFF" = 0) AND ("PREMIXING TRANSFER CYCLE DB".TRANSFER."TRANSFER BUFF"."PREMIXING TO STORAGE-4 WITH INLINE HOMO" = 0) AND ("PREMIXING DB"."MATERIAL SUCTION"."MATERIAL SUCTION BUFF" = 0) AND ("PREMIXING TRANSFER CYCLE DB".TRANSFER.SELECT."SELECT BUFF" = 3) AND ("CONTINUE DB"."PREMIXING PROCESS ERROR" <> 1) AND "PREMIXING TRANSFER CYCLE DB".TRANSFER."TRANSFER START" THEN
       "PREMIXING TRANSFER CYCLE DB".TRANSFER."TRANSFER BUFF"."PREMIXING TO STORAGE-4 WITH INLINE HOMO" := 5;
   END_IF;
END_REGION

REGION Network 18: WAIT
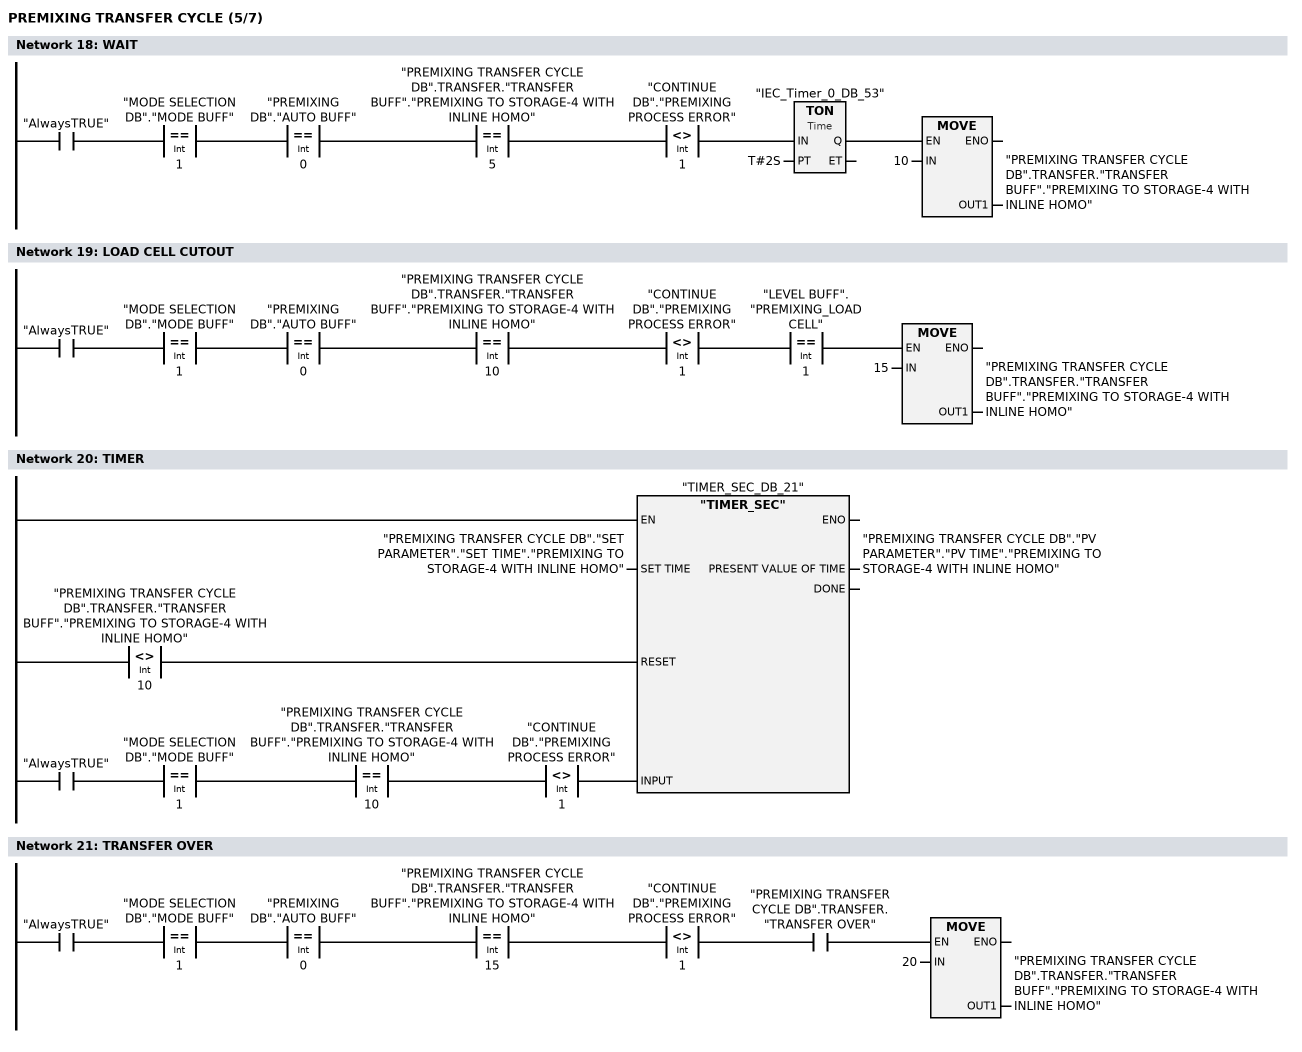
   RUNG wire#powerrail
      Contact( "AlwaysTRUE" )
      { S7_Templates := "SrcType := Int" } EQ_Contact(in1 := "MODE SELECTION DB"."MODE BUFF", in2 := 1)
      { S7_Templates := "SrcType := Int" } EQ_Contact(in1 := "PREMIXING DB"."AUTO BUFF", in2 := 0)
      { S7_Templates := "SrcType := Int" } EQ_Contact(in1 := "PREMIXING TRANSFER CYCLE DB".TRANSFER."TRANSFER BUFF"."PREMIXING TO STORAGE-4 WITH INLINE HOMO", in2 := 5)
      { S7_Templates := "SrcType := Int" } NE_Contact(in1 := "CONTINUE DB"."PREMIXING PROCESS ERROR", in2 := 1)
      { S7_Templates := "time_type := Time" } "IEC_Timer_0_DB_53".TON(pt := T#2S, et =>)
      Move(in := 10, out1 => "PREMIXING TRANSFER CYCLE DB".TRANSFER."TRANSFER BUFF"."PREMIXING TO STORAGE-4 WITH INLINE HOMO")
   END_RUNG
   // the same network as SCL:
   "IEC_Timer_0_DB_53".TON(IN := "AlwaysTRUE" AND ("MODE SELECTION DB"."MODE BUFF" = 1) AND ("PREMIXING DB"."AUTO BUFF" = 0) AND ("PREMIXING TRANSFER CYCLE DB".TRANSFER."TRANSFER BUFF"."PREMIXING TO STORAGE-4 WITH INLINE HOMO" = 5) AND ("CONTINUE DB"."PREMIXING PROCESS ERROR" <> 1),
                           PT := T#2S);
   IF "IEC_Timer_0_DB_53".Q THEN
       "PREMIXING TRANSFER CYCLE DB".TRANSFER."TRANSFER BUFF"."PREMIXING TO STORAGE-4 WITH INLINE HOMO" := 10;
   END_IF;
END_REGION

REGION Network 19: LOAD CELL CUTOUT
   RUNG wire#powerrail
      Contact( "AlwaysTRUE" )
      { S7_Templates := "SrcType := Int" } EQ_Contact(in1 := "MODE SELECTION DB"."MODE BUFF", in2 := 1)
      { S7_Templates := "SrcType := Int" } EQ_Contact(in1 := "PREMIXING DB"."AUTO BUFF", in2 := 0)
      { S7_Templates := "SrcType := Int" } EQ_Contact(in1 := "PREMIXING TRANSFER CYCLE DB".TRANSFER."TRANSFER BUFF"."PREMIXING TO STORAGE-4 WITH INLINE HOMO", in2 := 10)
      { S7_Templates := "SrcType := Int" } NE_Contact(in1 := "CONTINUE DB"."PREMIXING PROCESS ERROR", in2 := 1)
      { S7_Templates := "SrcType := Int" } EQ_Contact(in1 := "LEVEL BUFF"."PREMIXING_LOAD CELL", in2 := 1)
      Move(in := 15, out1 => "PREMIXING TRANSFER CYCLE DB".TRANSFER."TRANSFER BUFF"."PREMIXING TO STORAGE-4 WITH INLINE HOMO")
   END_RUNG
   // the same network as SCL:
   IF "AlwaysTRUE" AND ("MODE SELECTION DB"."MODE BUFF" = 1) AND ("PREMIXING DB"."AUTO BUFF" = 0) AND ("PREMIXING TRANSFER CYCLE DB".TRANSFER."TRANSFER BUFF"."PREMIXING TO STORAGE-4 WITH INLINE HOMO" = 10) AND ("CONTINUE DB"."PREMIXING PROCESS ERROR" <> 1) AND ("LEVEL BUFF"."PREMIXING_LOAD CELL" = 1) THEN
       "PREMIXING TRANSFER CYCLE DB".TRANSFER."TRANSFER BUFF"."PREMIXING TO STORAGE-4 WITH INLINE HOMO" := 15;
   END_IF;
END_REGION

REGION Network 20: TIMER
   RUNG wire#powerrail
      "TIMER_SEC_DB_21"(RESET := wire#w1, INPUT := wire#w2, "SET TIME" := "PREMIXING TRANSFER CYCLE DB"."SET PARAMETER"."SET TIME"."PREMIXING TO STORAGE-4 WITH INLINE HOMO", "PRESENT VALUE OF TIME" => "PREMIXING TRANSFER CYCLE DB"."PV PARAMETER"."PV TIME"."PREMIXING TO STORAGE-4 WITH INLINE HOMO", DONE =>)
   END_RUNG
   RUNG wire#powerrail
      { S7_Templates := "SrcType := Int" } NE_Contact(in1 := "PREMIXING TRANSFER CYCLE DB".TRANSFER."TRANSFER BUFF"."PREMIXING TO STORAGE-4 WITH INLINE HOMO", in2 := 10)
   END_RUNG wire#w1
   RUNG wire#powerrail
      Contact( "AlwaysTRUE" )
      { S7_Templates := "SrcType := Int" } EQ_Contact(in1 := "MODE SELECTION DB"."MODE BUFF", in2 := 1)
      { S7_Templates := "SrcType := Int" } EQ_Contact(in1 := "PREMIXING TRANSFER CYCLE DB".TRANSFER."TRANSFER BUFF"."PREMIXING TO STORAGE-4 WITH INLINE HOMO", in2 := 10)
      { S7_Templates := "SrcType := Int" } NE_Contact(in1 := "CONTINUE DB"."PREMIXING PROCESS ERROR", in2 := 1)
   END_RUNG wire#w2
   // the same network as SCL:
   "TIMER_SEC_DB_21"("SET TIME" := "PREMIXING TRANSFER CYCLE DB"."SET PARAMETER"."SET TIME"."PREMIXING TO STORAGE-4 WITH INLINE HOMO",   // "TIMER_SEC"
                     RESET := "PREMIXING TRANSFER CYCLE DB".TRANSFER."TRANSFER BUFF"."PREMIXING TO STORAGE-4 WITH INLINE HOMO" <> 10,
                     INPUT := "AlwaysTRUE" AND ("MODE SELECTION DB"."MODE BUFF" = 1) AND ("PREMIXING TRANSFER CYCLE DB".TRANSFER."TRANSFER BUFF"."PREMIXING TO STORAGE-4 WITH INLINE HOMO" = 10) AND ("CONTINUE DB"."PREMIXING PROCESS ERROR" <> 1),
                     "PRESENT VALUE OF TIME" => "PREMIXING TRANSFER CYCLE DB"."PV PARAMETER"."PV TIME"."PREMIXING TO STORAGE-4 WITH INLINE HOMO");
END_REGION

REGION Network 21: TRANSFER OVER
   RUNG wire#powerrail
      Contact( "AlwaysTRUE" )
      { S7_Templates := "SrcType := Int" } EQ_Contact(in1 := "MODE SELECTION DB"."MODE BUFF", in2 := 1)
      { S7_Templates := "SrcType := Int" } EQ_Contact(in1 := "PREMIXING DB"."AUTO BUFF", in2 := 0)
      { S7_Templates := "SrcType := Int" } EQ_Contact(in1 := "PREMIXING TRANSFER CYCLE DB".TRANSFER."TRANSFER BUFF"."PREMIXING TO STORAGE-4 WITH INLINE HOMO", in2 := 15)
      { S7_Templates := "SrcType := Int" } NE_Contact(in1 := "CONTINUE DB"."PREMIXING PROCESS ERROR", in2 := 1)
      Contact( "PREMIXING TRANSFER CYCLE DB".TRANSFER."TRANSFER OVER" )
      Move(in := 20, out1 => "PREMIXING TRANSFER CYCLE DB".TRANSFER."TRANSFER BUFF"."PREMIXING TO STORAGE-4 WITH INLINE HOMO")
   END_RUNG
   // the same network as SCL:
   IF "AlwaysTRUE" AND ("MODE SELECTION DB"."MODE BUFF" = 1) AND ("PREMIXING DB"."AUTO BUFF" = 0) AND ("PREMIXING TRANSFER CYCLE DB".TRANSFER."TRANSFER BUFF"."PREMIXING TO STORAGE-4 WITH INLINE HOMO" = 15) AND ("CONTINUE DB"."PREMIXING PROCESS ERROR" <> 1) AND "PREMIXING TRANSFER CYCLE DB".TRANSFER."TRANSFER OVER" THEN
       "PREMIXING TRANSFER CYCLE DB".TRANSFER."TRANSFER BUFF"."PREMIXING TO STORAGE-4 WITH INLINE HOMO" := 20;
   END_IF;
END_REGION

REGION Network 22: STOP
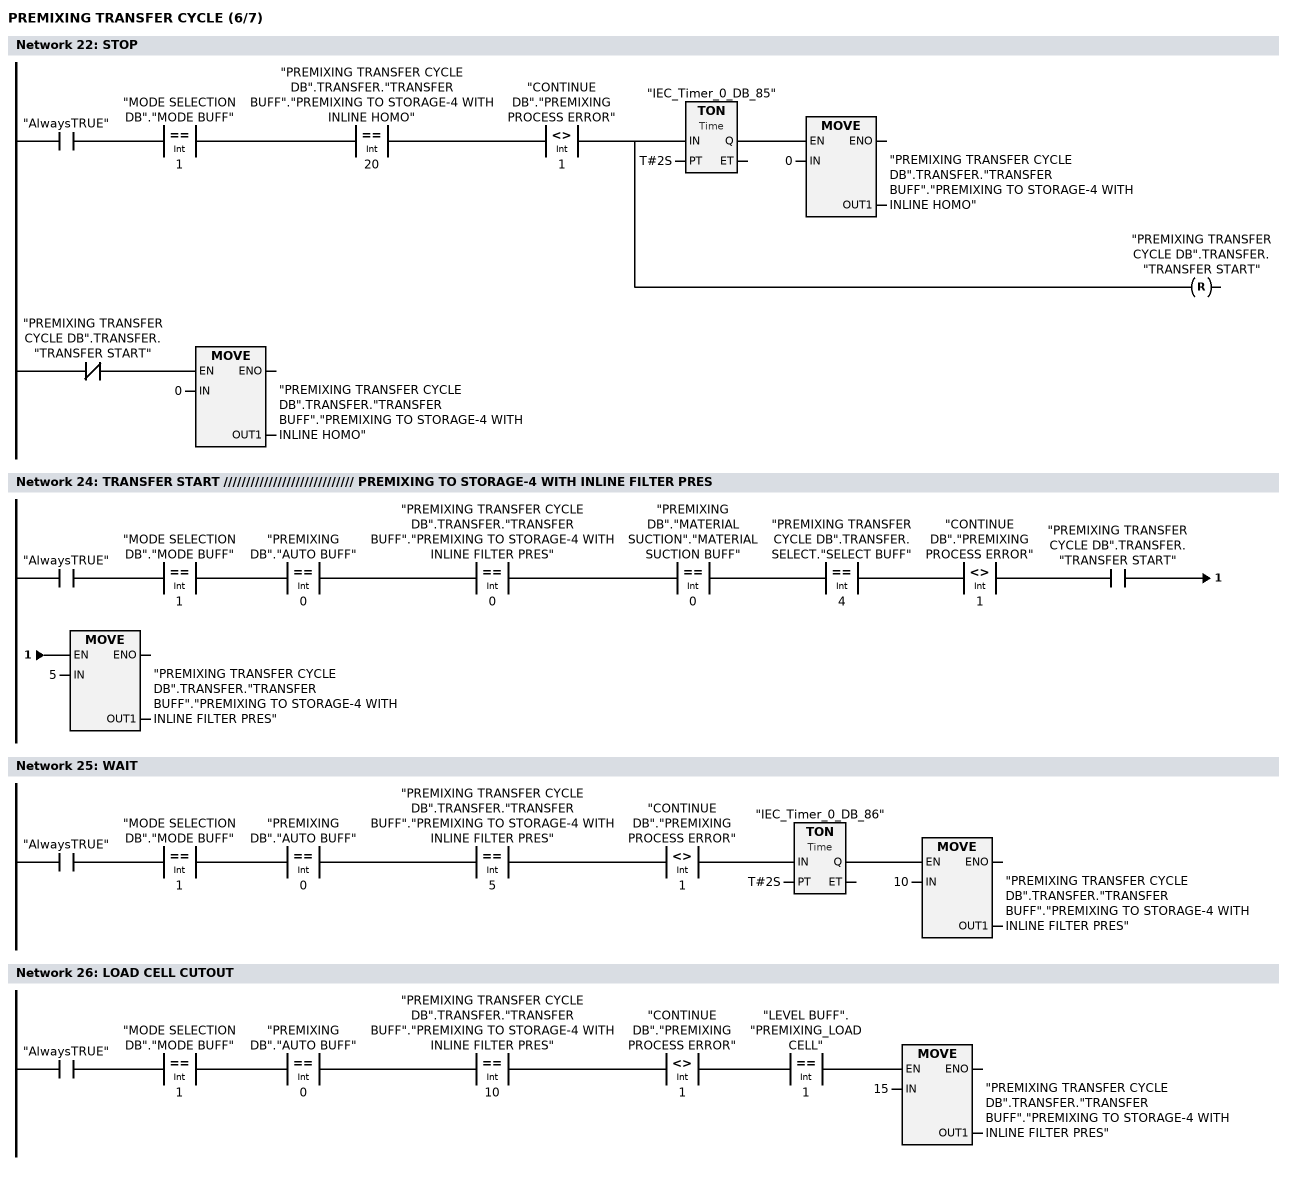
   RUNG wire#powerrail
      Contact( "AlwaysTRUE" )
      { S7_Templates := "SrcType := Int" } EQ_Contact(in1 := "MODE SELECTION DB"."MODE BUFF", in2 := 1)
      { S7_Templates := "SrcType := Int" } EQ_Contact(in1 := "PREMIXING TRANSFER CYCLE DB".TRANSFER."TRANSFER BUFF"."PREMIXING TO STORAGE-4 WITH INLINE HOMO", in2 := 20)
      { S7_Templates := "SrcType := Int" } NE_Contact(in1 := "CONTINUE DB"."PREMIXING PROCESS ERROR", in2 := 1)
      wire#w1
      { S7_Templates := "time_type := Time" } "IEC_Timer_0_DB_85".TON(pt := T#2S, et =>)
      Move(in := 0, out1 => "PREMIXING TRANSFER CYCLE DB".TRANSFER."TRANSFER BUFF"."PREMIXING TO STORAGE-4 WITH INLINE HOMO")
   END_RUNG
   RUNG wire#w1
      R_Coil( "PREMIXING TRANSFER CYCLE DB".TRANSFER."TRANSFER START" )
   END_RUNG
   RUNG wire#powerrail
      I_Contact( "PREMIXING TRANSFER CYCLE DB".TRANSFER."TRANSFER START" )
      Move(in := 0, out1 => "PREMIXING TRANSFER CYCLE DB".TRANSFER."TRANSFER BUFF"."PREMIXING TO STORAGE-4 WITH INLINE HOMO")
   END_RUNG
   // the same network as SCL:
   #_w1 := "AlwaysTRUE" AND ("MODE SELECTION DB"."MODE BUFF" = 1) AND ("PREMIXING TRANSFER CYCLE DB".TRANSFER."TRANSFER BUFF"."PREMIXING TO STORAGE-4 WITH INLINE HOMO" = 20) AND ("CONTINUE DB"."PREMIXING PROCESS ERROR" <> 1);
   "IEC_Timer_0_DB_85".TON(IN := #_w1, PT := T#2S);
   IF "IEC_Timer_0_DB_85".Q THEN
       "PREMIXING TRANSFER CYCLE DB".TRANSFER."TRANSFER BUFF"."PREMIXING TO STORAGE-4 WITH INLINE HOMO" := 0;
   END_IF;
   IF #_w1 THEN "PREMIXING TRANSFER CYCLE DB".TRANSFER."TRANSFER START" := FALSE; END_IF;
   IF NOT "PREMIXING TRANSFER CYCLE DB".TRANSFER."TRANSFER START" THEN
       "PREMIXING TRANSFER CYCLE DB".TRANSFER."TRANSFER BUFF"."PREMIXING TO STORAGE-4 WITH INLINE HOMO" := 0;
   END_IF;
END_REGION

REGION Network 24: TRANSFER START ///////////////////////////// PREMIXING TO STORAGE-4 WITH INLINE FILTER PRES
   RUNG wire#powerrail
      Contact( "AlwaysTRUE" )
      { S7_Templates := "SrcType := Int" } EQ_Contact(in1 := "MODE SELECTION DB"."MODE BUFF", in2 := 1)
      { S7_Templates := "SrcType := Int" } EQ_Contact(in1 := "PREMIXING DB"."AUTO BUFF", in2 := 0)
      { S7_Templates := "SrcType := Int" } EQ_Contact(in1 := "PREMIXING TRANSFER CYCLE DB".TRANSFER."TRANSFER BUFF"."PREMIXING TO STORAGE-4 WITH INLINE FILTER PRES", in2 := 0)
      { S7_Templates := "SrcType := Int" } EQ_Contact(in1 := "PREMIXING DB"."MATERIAL SUCTION"."MATERIAL SUCTION BUFF", in2 := 0)
      { S7_Templates := "SrcType := Int" } EQ_Contact(in1 := "PREMIXING TRANSFER CYCLE DB".TRANSFER.SELECT."SELECT BUFF", in2 := 4)
      { S7_Templates := "SrcType := Int" } NE_Contact(in1 := "CONTINUE DB"."PREMIXING PROCESS ERROR", in2 := 1)
      Contact( "PREMIXING TRANSFER CYCLE DB".TRANSFER."TRANSFER START" )
      Move(in := 5, out1 => "PREMIXING TRANSFER CYCLE DB".TRANSFER."TRANSFER BUFF"."PREMIXING TO STORAGE-4 WITH INLINE FILTER PRES")
   END_RUNG
   // the same network as SCL:
   IF "AlwaysTRUE" AND ("MODE SELECTION DB"."MODE BUFF" = 1) AND ("PREMIXING DB"."AUTO BUFF" = 0) AND ("PREMIXING TRANSFER CYCLE DB".TRANSFER."TRANSFER BUFF"."PREMIXING TO STORAGE-4 WITH INLINE FILTER PRES" = 0) AND ("PREMIXING DB"."MATERIAL SUCTION"."MATERIAL SUCTION BUFF" = 0) AND ("PREMIXING TRANSFER CYCLE DB".TRANSFER.SELECT."SELECT BUFF" = 4) AND ("CONTINUE DB"."PREMIXING PROCESS ERROR" <> 1) AND "PREMIXING TRANSFER CYCLE DB".TRANSFER."TRANSFER START" THEN
       "PREMIXING TRANSFER CYCLE DB".TRANSFER."TRANSFER BUFF"."PREMIXING TO STORAGE-4 WITH INLINE FILTER PRES" := 5;
   END_IF;
END_REGION

REGION Network 25: WAIT
   RUNG wire#powerrail
      Contact( "AlwaysTRUE" )
      { S7_Templates := "SrcType := Int" } EQ_Contact(in1 := "MODE SELECTION DB"."MODE BUFF", in2 := 1)
      { S7_Templates := "SrcType := Int" } EQ_Contact(in1 := "PREMIXING DB"."AUTO BUFF", in2 := 0)
      { S7_Templates := "SrcType := Int" } EQ_Contact(in1 := "PREMIXING TRANSFER CYCLE DB".TRANSFER."TRANSFER BUFF"."PREMIXING TO STORAGE-4 WITH INLINE FILTER PRES", in2 := 5)
      { S7_Templates := "SrcType := Int" } NE_Contact(in1 := "CONTINUE DB"."PREMIXING PROCESS ERROR", in2 := 1)
      { S7_Templates := "time_type := Time" } "IEC_Timer_0_DB_86".TON(pt := T#2S, et =>)
      Move(in := 10, out1 => "PREMIXING TRANSFER CYCLE DB".TRANSFER."TRANSFER BUFF"."PREMIXING TO STORAGE-4 WITH INLINE FILTER PRES")
   END_RUNG
   // the same network as SCL:
   "IEC_Timer_0_DB_86".TON(IN := "AlwaysTRUE" AND ("MODE SELECTION DB"."MODE BUFF" = 1) AND ("PREMIXING DB"."AUTO BUFF" = 0) AND ("PREMIXING TRANSFER CYCLE DB".TRANSFER."TRANSFER BUFF"."PREMIXING TO STORAGE-4 WITH INLINE FILTER PRES" = 5) AND ("CONTINUE DB"."PREMIXING PROCESS ERROR" <> 1),
                           PT := T#2S);
   IF "IEC_Timer_0_DB_86".Q THEN
       "PREMIXING TRANSFER CYCLE DB".TRANSFER."TRANSFER BUFF"."PREMIXING TO STORAGE-4 WITH INLINE FILTER PRES" := 10;
   END_IF;
END_REGION

REGION Network 26: LOAD CELL CUTOUT
   RUNG wire#powerrail
      Contact( "AlwaysTRUE" )
      { S7_Templates := "SrcType := Int" } EQ_Contact(in1 := "MODE SELECTION DB"."MODE BUFF", in2 := 1)
      { S7_Templates := "SrcType := Int" } EQ_Contact(in1 := "PREMIXING DB"."AUTO BUFF", in2 := 0)
      { S7_Templates := "SrcType := Int" } EQ_Contact(in1 := "PREMIXING TRANSFER CYCLE DB".TRANSFER."TRANSFER BUFF"."PREMIXING TO STORAGE-4 WITH INLINE FILTER PRES", in2 := 10)
      { S7_Templates := "SrcType := Int" } NE_Contact(in1 := "CONTINUE DB"."PREMIXING PROCESS ERROR", in2 := 1)
      { S7_Templates := "SrcType := Int" } EQ_Contact(in1 := "LEVEL BUFF"."PREMIXING_LOAD CELL", in2 := 1)
      Move(in := 15, out1 => "PREMIXING TRANSFER CYCLE DB".TRANSFER."TRANSFER BUFF"."PREMIXING TO STORAGE-4 WITH INLINE FILTER PRES")
   END_RUNG
   // the same network as SCL:
   IF "AlwaysTRUE" AND ("MODE SELECTION DB"."MODE BUFF" = 1) AND ("PREMIXING DB"."AUTO BUFF" = 0) AND ("PREMIXING TRANSFER CYCLE DB".TRANSFER."TRANSFER BUFF"."PREMIXING TO STORAGE-4 WITH INLINE FILTER PRES" = 10) AND ("CONTINUE DB"."PREMIXING PROCESS ERROR" <> 1) AND ("LEVEL BUFF"."PREMIXING_LOAD CELL" = 1) THEN
       "PREMIXING TRANSFER CYCLE DB".TRANSFER."TRANSFER BUFF"."PREMIXING TO STORAGE-4 WITH INLINE FILTER PRES" := 15;
   END_IF;
END_REGION

REGION Network 27: TIMER
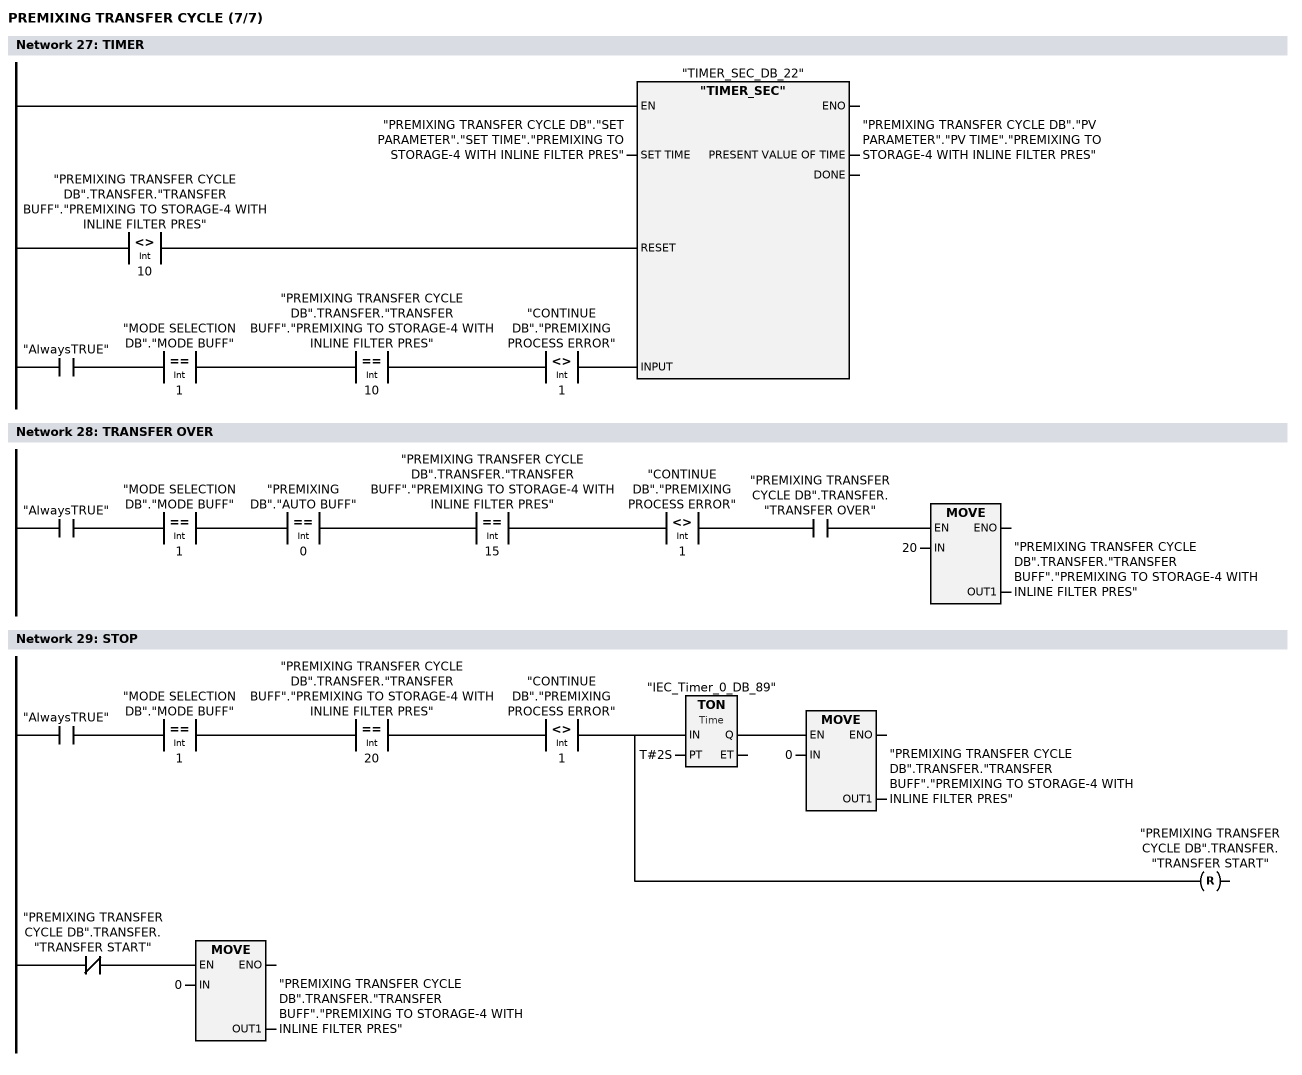
   RUNG wire#powerrail
      "TIMER_SEC_DB_22"(RESET := wire#w1, INPUT := wire#w2, "SET TIME" := "PREMIXING TRANSFER CYCLE DB"."SET PARAMETER"."SET TIME"."PREMIXING TO STORAGE-4 WITH INLINE FILTER PRES", "PRESENT VALUE OF TIME" => "PREMIXING TRANSFER CYCLE DB"."PV PARAMETER"."PV TIME"."PREMIXING TO STORAGE-4 WITH INLINE FILTER PRES", DONE =>)
   END_RUNG
   RUNG wire#powerrail
      { S7_Templates := "SrcType := Int" } NE_Contact(in1 := "PREMIXING TRANSFER CYCLE DB".TRANSFER."TRANSFER BUFF"."PREMIXING TO STORAGE-4 WITH INLINE FILTER PRES", in2 := 10)
   END_RUNG wire#w1
   RUNG wire#powerrail
      Contact( "AlwaysTRUE" )
      { S7_Templates := "SrcType := Int" } EQ_Contact(in1 := "MODE SELECTION DB"."MODE BUFF", in2 := 1)
      { S7_Templates := "SrcType := Int" } EQ_Contact(in1 := "PREMIXING TRANSFER CYCLE DB".TRANSFER."TRANSFER BUFF"."PREMIXING TO STORAGE-4 WITH INLINE FILTER PRES", in2 := 10)
      { S7_Templates := "SrcType := Int" } NE_Contact(in1 := "CONTINUE DB"."PREMIXING PROCESS ERROR", in2 := 1)
   END_RUNG wire#w2
   // the same network as SCL:
   "TIMER_SEC_DB_22"("SET TIME" := "PREMIXING TRANSFER CYCLE DB"."SET PARAMETER"."SET TIME"."PREMIXING TO STORAGE-4 WITH INLINE FILTER PRES",   // "TIMER_SEC"
                     RESET := "PREMIXING TRANSFER CYCLE DB".TRANSFER."TRANSFER BUFF"."PREMIXING TO STORAGE-4 WITH INLINE FILTER PRES" <> 10,
                     INPUT := "AlwaysTRUE" AND ("MODE SELECTION DB"."MODE BUFF" = 1) AND ("PREMIXING TRANSFER CYCLE DB".TRANSFER."TRANSFER BUFF"."PREMIXING TO STORAGE-4 WITH INLINE FILTER PRES" = 10) AND ("CONTINUE DB"."PREMIXING PROCESS ERROR" <> 1),
                     "PRESENT VALUE OF TIME" => "PREMIXING TRANSFER CYCLE DB"."PV PARAMETER"."PV TIME"."PREMIXING TO STORAGE-4 WITH INLINE FILTER PRES");
END_REGION

REGION Network 28: TRANSFER OVER
   RUNG wire#powerrail
      Contact( "AlwaysTRUE" )
      { S7_Templates := "SrcType := Int" } EQ_Contact(in1 := "MODE SELECTION DB"."MODE BUFF", in2 := 1)
      { S7_Templates := "SrcType := Int" } EQ_Contact(in1 := "PREMIXING DB"."AUTO BUFF", in2 := 0)
      { S7_Templates := "SrcType := Int" } EQ_Contact(in1 := "PREMIXING TRANSFER CYCLE DB".TRANSFER."TRANSFER BUFF"."PREMIXING TO STORAGE-4 WITH INLINE FILTER PRES", in2 := 15)
      { S7_Templates := "SrcType := Int" } NE_Contact(in1 := "CONTINUE DB"."PREMIXING PROCESS ERROR", in2 := 1)
      Contact( "PREMIXING TRANSFER CYCLE DB".TRANSFER."TRANSFER OVER" )
      Move(in := 20, out1 => "PREMIXING TRANSFER CYCLE DB".TRANSFER."TRANSFER BUFF"."PREMIXING TO STORAGE-4 WITH INLINE FILTER PRES")
   END_RUNG
   // the same network as SCL:
   IF "AlwaysTRUE" AND ("MODE SELECTION DB"."MODE BUFF" = 1) AND ("PREMIXING DB"."AUTO BUFF" = 0) AND ("PREMIXING TRANSFER CYCLE DB".TRANSFER."TRANSFER BUFF"."PREMIXING TO STORAGE-4 WITH INLINE FILTER PRES" = 15) AND ("CONTINUE DB"."PREMIXING PROCESS ERROR" <> 1) AND "PREMIXING TRANSFER CYCLE DB".TRANSFER."TRANSFER OVER" THEN
       "PREMIXING TRANSFER CYCLE DB".TRANSFER."TRANSFER BUFF"."PREMIXING TO STORAGE-4 WITH INLINE FILTER PRES" := 20;
   END_IF;
END_REGION

REGION Network 29: STOP
   RUNG wire#powerrail
      Contact( "AlwaysTRUE" )
      { S7_Templates := "SrcType := Int" } EQ_Contact(in1 := "MODE SELECTION DB"."MODE BUFF", in2 := 1)
      { S7_Templates := "SrcType := Int" } EQ_Contact(in1 := "PREMIXING TRANSFER CYCLE DB".TRANSFER."TRANSFER BUFF"."PREMIXING TO STORAGE-4 WITH INLINE FILTER PRES", in2 := 20)
      { S7_Templates := "SrcType := Int" } NE_Contact(in1 := "CONTINUE DB"."PREMIXING PROCESS ERROR", in2 := 1)
      wire#w1
      { S7_Templates := "time_type := Time" } "IEC_Timer_0_DB_89".TON(pt := T#2S, et =>)
      Move(in := 0, out1 => "PREMIXING TRANSFER CYCLE DB".TRANSFER."TRANSFER BUFF"."PREMIXING TO STORAGE-4 WITH INLINE FILTER PRES")
   END_RUNG
   RUNG wire#w1
      R_Coil( "PREMIXING TRANSFER CYCLE DB".TRANSFER."TRANSFER START" )
   END_RUNG
   RUNG wire#powerrail
      I_Contact( "PREMIXING TRANSFER CYCLE DB".TRANSFER."TRANSFER START" )
      Move(in := 0, out1 => "PREMIXING TRANSFER CYCLE DB".TRANSFER."TRANSFER BUFF"."PREMIXING TO STORAGE-4 WITH INLINE FILTER PRES")
   END_RUNG
   // the same network as SCL:
   #_w1 := "AlwaysTRUE" AND ("MODE SELECTION DB"."MODE BUFF" = 1) AND ("PREMIXING TRANSFER CYCLE DB".TRANSFER."TRANSFER BUFF"."PREMIXING TO STORAGE-4 WITH INLINE FILTER PRES" = 20) AND ("CONTINUE DB"."PREMIXING PROCESS ERROR" <> 1);
   "IEC_Timer_0_DB_89".TON(IN := #_w1, PT := T#2S);
   IF "IEC_Timer_0_DB_89".Q THEN
       "PREMIXING TRANSFER CYCLE DB".TRANSFER."TRANSFER BUFF"."PREMIXING TO STORAGE-4 WITH INLINE FILTER PRES" := 0;
   END_IF;
   IF #_w1 THEN "PREMIXING TRANSFER CYCLE DB".TRANSFER."TRANSFER START" := FALSE; END_IF;
   IF NOT "PREMIXING TRANSFER CYCLE DB".TRANSFER."TRANSFER START" THEN
       "PREMIXING TRANSFER CYCLE DB".TRANSFER."TRANSFER BUFF"."PREMIXING TO STORAGE-4 WITH INLINE FILTER PRES" := 0;
   END_IF;
END_REGION
END_FUNCTION
